// TIA Portal V18 export
TYPE "LGasp_typeCmdManAttuatore"
// stored: IsFailsafeCompliant false
   STRUCT
      startcicloman : Bool;   // Cmd start --> posizionamento se asse , ciclo stampo se EV
      jogpos : Bool;   // Cmd jog positivo
      jogneg : Bool;   // Cmd jog negativo
   END_STRUCT;
END_TYPE
